FUNCTION_BLOCK FB_EK1100
VAR_OUTPUT
	state						AT %I* : UINT;
END_VAR

END_FUNCTION_BLOCK

(* stored: Version 1.1.0.1, ProductVersion 3.1.4026.18
   POU FB_EK1100: Id {f0915f53-deb0-41a0-9767-43d19234ebbf}, SpecialFunc None *)
